PROGRAM MAIN
VAR
END_VAR

.Global_Variables.TcJoy();

IF .Global_Variables.TcJoy.bIsActive THEN
	;
END_IF

END_PROGRAM

(* stored: Version 1.1.0.1, ProductVersion 3.1.4024.3
   POU MAIN: Id {d25881fd-bae0-4e0a-b3eb-c173027ef094}, SpecialFunc None *)
